(* IEC 61131-3 sources: inproshop/test14_exported/OP11/1.Global, 7 files *)

(* ---- DB1100_Control.st ---- *)
VAR_GLOBAL
	Mode:Str_Mode;
	HMI:Str_HMI;
END_VAR
VAR_GLOBAL RETAIN PERSISTENT
	Machine AT %MB132276 : Str_Machine;
END_VAR

(* ---- DB1102_Recipe.st ---- *)
VAR_GLOBAL
END_VAR
VAR_GLOBAL RETAIN PERSISTENT

	RecipeChangePmt AT %MB132596 : BOOL;	//配方允许切换
	ParameterChangePmt AT %MB132597 : BOOL;	//参数允许更改
	RecipeNumTemp AT %MB132598 : INT;	//HMI选中还未保存到PLC的编号.
	RecipeNum AT %MB132600 : INT;	//配方元素编号.
	RecipeName AT %MB133699 : STRING(20);	//配方元素名称.
	RecipeNameTemp AT %MB133720 : STRING(20);	//HMI头部显示当前配方名称
	RecipeOk AT %MB132602 : BOOL;//配方可用
	DownLoad AT %MB132603 : BOOL;//配方下载
	TypeDataCur AT %MB146576 : Str_OP11_Recipe;//当前配方
	TypeData AT %MB305052 : ARRAY [0..20] OF Str_OP11_Recipe;//配方数据
END_VAR

(* ---- DB1103_Count.st ---- *)
VAR_GLOBAL RETAIN PERSISTENT
	Total AT %MB145904 : Str_Count;//总计数
	OK AT %MB174656 : Str_Count;//OK计数
	NG AT %MB175328 : Str_Count;//NG计数
END_VAR
VAR_GLOBAL
	Yield : REAL;//良品率
	Clear : BOOL;//清除计数
END_VAR

(* ---- DB1105_Communication.st ---- *)
VAR_GLOBAL
	TcpClient:ARRAY[0..9] OF Str_TcpClient;
	TcpSever:ARRAY[0..9] OF Str_TcpClient;
	From_OPXX    :Str_OP80_TO_OPXX;
	TO_OPXX    :Str_OPXX_TO_OP80;
	FromMaster  :Str_FromMaster;
END_VAR

(* ---- DB1150_DriveControl.st ---- *)
VAR_GLOBAL RETAIN PERSISTENT
	CylCtrl AT %MB288288 : ARRAY [0..63] OF Str_Cylinder;
	VacCtrl AT %MB296864 : ARRAY [0..32] OF Str_Cylinder;
	AxisCtrl AT %MB341036 : ARRAY [0..16] OF Str_Axis;
	Sensor AT %MB301288 : ARRAY [0..32] OF Str_Sensor;
	CamCtrl AT %MB133684 : ARRAY [1..3] OF Str_CamControl;
END_VAR

VAR_GLOBAL
	DoubleStart:ARRAY [1..4] OF Str_DoubleStart;
	Epson : ARRAY [1..10] OF Str_Epson;
	Kuka : ARRAY [1..2] OF Str_Kuka6;
	Rotdisk:ARRAY [1..1] OF Str_Rotdisk;
	Stopper:ARRAY [1..20] OF Str_Stopper;
	Motor:ARRAY [1..10] OF Str_Motor;
	AI:ARRAY [0..200] OF Str_AI;
	AAS:ARRAY [1..1] OF Str_AAS;
	HeatCtrl : ARRAY [1..1] OF Str_Heating;
	PalletCtrl : ARRAY [0..3] OF Str_Palletizing;
END_VAR

(* ---- DB1170_Fault.st ---- *)
VAR_GLOBAL
	Estop:Str_OP11_FaultEstop;//紧急停止类报警
	Stop:Str_OP11_Faultstop;//暂停类报警
	Run:Str_OP11_FaultRun;//警告类报警
	EstopTotal:BOOL;//急停报警汇总
	StopTotal:BOOL;//暂停报警汇总
	RunTotal:BOOL;//警告汇总
END_VAR

(* ---- DB1190_Other.st ---- *)
VAR_GLOBAL RETAIN PERSISTENT
	{attribute 'ElemComment':='(),(上料机械臂取料夹爪),(上料机械臂放料夹爪),(缓存台1),(缓存台2),(缓存台3),(缓存台4),(测试台1),(测试台2),(测试台3),(测试台4),(下料机械臂),4()'}
	StationData AT %MB305600 : ARRAY [0..15] OF Str_OP11_StationData;
END_VAR
